{attribute addProperty BoxType "BK1120-0000-0001"}
{attribute addProperty Id "Term_375_KL1002KL1002_D229A9CA00"}
{attribute addProperty CRC "1821467411"}
{attribute addProperty SizeInBites "0"}
{attribute addProperty SizeInBytes "0"}
TYPE A_0002_BK1120_0000_0001_6C916313 EXTENDS BK1120_4487A81F :
STRUCT
	{attribute addProperty Name "Term_375_KL1002"}
	Term_375_KL1002 : KL1002_D229A9CA;
END_STRUCT
END_TYPE

(* stored: Version 1.2.0.0, ProductVersion 3.1.4024.9
   DUT A_0002_BK1120_0000_0001_6C916313: Id {7c87e29e-97a9-4f39-be39-6b927bece357} *)
